FUNCTION_BLOCK FB_TestHTTP_Get_openWeatherMap
VAR_INPUT
    bSend             : BOOL;
END_VAR
VAR_IN_OUT
    fbClient          : FB_IotHttpClient;
END_VAR
VAR_OUTPUT
    bBusy             : BOOL;
    bError            : BOOL;
END_VAR
VAR
    fbRequest         : FB_IotHttpRequest;
    fbJson            : FB_JsonDomParser;
    nState            : UDINT;
    RisingEdge        : R_TRIG;

    bGetContentResult : BOOL;
    sContent          : STRING(511);

    bGetJsonResult    : BOOL;
    jsonDoc           : SJsonValue;
    jsonVal           : SJsonValue;
    sResultValue      : STRING;

    nReqCount         : UDINT;
    nResCount         : UDINT;
    nValidResCount    : UDINT;
    nErrCount         : UDINT;
	
	// split string
	aSplit					:ARRAY[0..cMax] OF STRING(255);
	bResultSplit			:BOOL;
	ii						:UDINT;
END_VAR
VAR CONSTANT
	cMax					:UDINT := 15;
END_VAR

RisingEdge(CLK:= bSend);
CASE nState OF
0:
    IF RisingEdge.Q THEN
        IF fbRequest.SendRequest(sUri:= '/repos/ECCO-RUO/test-branches-config-file/tags',
                                 fbClient:= fbClient, 
                                 eRequestType:= ETcIotHttpRequestType.HTTP_Get, 0, 0, 0) THEN
            nState:= 1;
            nReqCount:= nReqCount+1;
            bBusy:= TRUE;
            bError:= FALSE;
        END_IF
    END_IF
1:
    IF NOT fbRequest.bBusy THEN
        bError:= TRUE;
        IF NOT fbRequest.bError THEN
            bGetContentResult:= fbRequest.GetContent(pContent:= ADR(sContent), 
                                                     nContentSize:= SIZEOF(sContent), 
                                                     bSetNullTermination:= TRUE);
            IF fbRequest.nStatusCode >= 200 AND fbRequest.nStatusCode < 300 THEN
                bGetJsonResult:= FALSE;
                jsonDoc:= fbRequest.GetJsonDomContent(fbJson);
                IF jsonDoc <> 0 THEN
					
					//do something with the weather data
//                    GVL.sVars.sTag := sContent;
					// split/parse strings
					FOR ii := 0 TO cMax - 1 DO
						
						aSplit[ii] := sContent;
						bResultSplit := FindAndSplitChar(sSeparatorChar := '"', pSrcString := ADR(aSplit[ii]),
														  pLeftString := ADR(aSplit[ii + 1]), nLeftSize := SIZEOF(aSplit[ii + 1]),
														  pRightString := ADR(aSplit[ii]), nRightSize := SIZEOF(aSplit[ii]),
														  bSearchFromRight := FALSE);
														  
						// assign values from config file
						GVL.sVars.sEnvironment		:= aSplit[0];
						
						IF NOT bResultSplit THEN
							EXIT;
						END_IF
					END_FOR
					
					nValidResCount:= nValidResCount+1;
                    bError:= FALSE;
                END_IF
                nResCount:= nResCount+1;
            END_IF
        END_IF
        nState:= 0;
        bBusy:= FALSE;
        IF bError THEN
            nErrCount:= nErrCount+1;
        END_IF
    END_IF
END_CASE

END_FUNCTION_BLOCK

(* stored: Version 1.1.0.1, ProductVersion 3.1.4024.6
   POU FB_TestHTTP_Get_openWeatherMap: Id {eca3dfed-7a20-454d-89af-a713fb3d59c6}, SpecialFunc None *)
